(********************* G.D S.p.A. - Technical Department ***********************************
This program has been generated automatically from Application Designer DE&F
********************************************************************************************)
PROGRAM dbg_csp_transfer_crosspusher_sensors
VAR
  high_achk_shd : analog_check_shadow;
  high_ai_shd : analog_input_shadow;
END_VAR

_objects_manager();

IF	g_application_status <> APPLICATION_STATUS_RUNNING
THEN
	RETURN;
END_IF

CASE process_get_mode(CONVERSION_this := dbg_root.prc) OF
	MODE_ABSENT,
	MODE_INACTIVE:
		RETURN;
	MODE_TEST:
		RETURN;
END_CASE

ACTION _objects_manager:
IF	objects_initialization()
THEN


	RETURN;
END_IF

IF	objects_running()
THEN
;
END_IF
END_ACTION

END_PROGRAM

(* stored: Version 1.1.0.1, ProductVersion 3.1.4024.3
   POU dbg_csp_transfer_crosspusher_sensors: Id {6fd05283-1772-43f7-88f8-b1a736a8c979}, SpecialFunc None
   Action _objects_manager: Id {d49dd11f-fd04-49a0-8466-22370fc4df46} *)
